FUNCTION_BLOCK MoverList EXTENDS Objective
VAR_INPUT
END_VAR
VAR_OUTPUT
END_VAR
VAR
END_VAR

METHOD MoveAllToPosition : MoverList
VAR_INPUT

	DestinationPosition		: LREAL;		// position on track for all shuttles to move towards	

END_VAR

VAR
	i: USINT;
END_VAR

// For every valid mover in the list, pass it a MoveToPosition command
FOR i := 0 TO SIZEOF( THIS^.TrackedMovers ) / SIZEOF( THIS^.TrackedMovers[i] ) - 1 DO
	
	IF THIS^.TrackedMovers[i] <> 0 THEN
		THIS^.TrackedMovers[i]^.MoveToPosition( DestinationPosition );
	END_IF

END_FOR
END_METHOD

METHOD MoveAllToStation : MoverList
VAR_INPUT
	
	DestinationStation	: REFERENCE TO Station;

END_VAR

VAR
	i : USINT;
END_VAR

// For every valid mover in the list, pass it a MoveToStation command
FOR i := 0 TO SIZEOF( THIS^.TrackedMovers ) / SIZEOF( THIS^.TrackedMovers[i] ) - 1 DO
	
	IF THIS^.TrackedMovers[i] <> 0 THEN
		THIS^.TrackedMovers[i]^.MoveToStation( DestinationStation ) ;
	END_IF

END_FOR
END_METHOD

METHOD SetAllAcceleration : MoverList
VAR_INPUT
	
	Acceleration		: LREAL;

END_VAR

VAR
	i	: USINT;
END_VAR

// For every valid mover in the list, set the Acceleration values
FOR i := 0 TO SIZEOF( THIS^.TrackedMovers ) / SIZEOF( THIS^.TrackedMovers[i] ) - 1 DO
	
	IF THIS^.TrackedMovers[i] <> 0 THEN
		THIS^.TrackedMovers[i]^.SetAcceleration( Acceleration );
	END_IF

END_FOR
END_METHOD

METHOD SetAllDeceleration : MoverList
VAR_INPUT
	
	Deceleration		: LREAL;
	
END_VAR
VAR
	i	: USINT;
END_VAR

// For every valid mover in the list, set the Deceleration values
FOR i := 0 TO SIZEOF( THIS^.TrackedMovers ) / SIZEOF( THIS^.TrackedMovers[i] ) - 1 DO
	
	IF THIS^.TrackedMovers[i] <> 0 THEN
		THIS^.TrackedMovers[i]^.SetDeceleration( Deceleration );
	END_IF

END_FOR
END_METHOD

METHOD SetAllVelocity : MoverList
VAR_INPUT
	
	Velocity	: LREAL;	

END_VAR
VAR
	i	: USINT;
END_VAR

// For every valid mover in the list, set the Velocity values
FOR i := 0 TO SIZEOF( THIS^.TrackedMovers ) / SIZEOF( THIS^.TrackedMovers[i] ) - 1 DO
	
	IF THIS^.TrackedMovers[i] <> 0 THEN
		THIS^.TrackedMovers[i]^.SetVelocity( Velocity );
	END_IF

END_FOR
END_METHOD

METHOD StopAll : MoverList
VAR_INPUT
END_VAR

VAR
	i	: USINT;
END_VAR


// Stop all valid movers in the list
FOR i := 0 TO SIZEOF( THIS^.TrackedMovers ) / SIZEOF( THIS^.TrackedMovers[i] ) - 1 DO
	
	IF THIS^.TrackedMovers[i] <> 0 THEN
		THIS^.TrackedMovers[i]^.Stop();
	END_IF

END_FOR
END_METHOD

METHOD UnregisterAll : BOOL
VAR_INPUT
END_VAR
VAR
	i	: USINT;
END_VAR


FOR i := 0 TO SIZEOF( THIS^.TrackedMovers ) / SIZEOF( THIS^.TrackedMovers[i] ) - 1 DO
	IF THIS^.TrackedMovers[i] <> 0 THEN
		THIS^.UnregisterMover( THIS^.TrackedMovers[i]^ );
	END_IF
END_FOR
END_METHOD

END_FUNCTION_BLOCK

(* stored: Version 1.1.0.1, ProductVersion 3.1.4024.9
   POU MoverList: Id {6a6492c3-5dac-4c49-8708-8eab34cf4a1d}, SpecialFunc None
   Folder Methods: Id {f0610894-1931-4d0e-a817-1d1b4c8212b1}
   Folder Properties: Id {3fdda14a-1516-48f6-a734-917962304085}
   Method MoveAllToPosition: Id {bd912cae-8475-45f4-9366-6d4e3f45dbfd}
   Method MoveAllToStation: Id {7e8649c5-afae-438c-9d7c-0849d9778d85}
   Method SetAllAcceleration: Id {e13ce26b-c052-44c4-b781-edc2323e6bd8}
   Method SetAllDeceleration: Id {b4a74589-da0f-40fe-9d74-9df176d68d9e}
   Method SetAllVelocity: Id {cee9569c-3982-4955-90f1-8e5baf09c135}
   Method StopAll: Id {52e8beec-48ea-4912-8399-13b65c4fd5d8}
   Method UnregisterAll: Id {9f7a3d8e-3975-4fa4-8579-c54f77146104} *)
